// TIA Portal V19 export
ORGANIZATION_BLOCK "IO access error"   // OB122, STL, IOAccessError
{ S7_Optimized_Access := 'FALSE' }
   VAR_TEMP
      EV_CLASS : Byte;   // 16#29: Event class 2, Entering event state, Internal fault event
      SW_FLT : Byte;   // 16#42:reading, 16#43:writing
      PRIORITY : Byte;   // Priority of OB Execution
      OB_NUMBR : Byte;   // OB number
      BLK_TYPE : Byte;   // 16#88:OB, 16#8C:FC, 16#8E:FB: Type of block causing the error
      MEM_AREA : Byte;   // Memory area and access type
      MEM_ADDR : Word;   // Memory address where access error occured
      BLK_NUM : Word;   // Block number in which error occured
      PRG_ADDR : Word;   // Program address where error occured
      DATE_TIME : Date_And_Time;   // Date and time OB started
   END_VAR
BEGIN
END_ORGANIZATION_BLOCK
